FUNCTION_BLOCK XtsHardware
VAR_INPUT
END_VAR
VAR_OUTPUT
	XtsHardwareOK : BOOL;
	Xts48VStanding : BOOL;
	Xts24VStanding : BOOL;
END_VAR
VAR
	XtsIoEnvironment : Tc3_XTS_Utility.FB_TcIoXtsEnvironment;
	bInit: BOOL;
	bMoverIdDetectionError		: BOOL;
	bMoverIdDetectionActive		: BOOL;
	bMoverIdDetected : BOOL;
	f24V: ARRAY[1..nModuleNumber] OF LREAL;
	f48V: ARRAY[1..nModuleNumber] OF LREAL;
	CurrentLive : ARRAY[1..nModuleNumber] OF LREAL;
	MaxCurrent : ARRAY [1..nModuleNumber] OF DINT;
	nModuleCounter : INT := 1;
	nForCounter1 : UDINT;
	i: INT;
	State :(
        Init,                                               
		Redetect,
		MoversValid,                                 
        AllMoversFound,
		MoverIdDetection,
		XTSMode,
		CheckModuleVoltages,
		HWReady);
	Logger : TcMessage_Ext;
END_VAR
VAR CONSTANT
	nModuleNumber  : INT := 16;
END_VAR

IF NOT bInit THEN
	IF XtsIoEnvironment.Init(TRUE) THEN
		XtsIoEnvironment.Init(FALSE);
		bInit := TRUE;
	END_IF
	RETURN;
END_IF

CASE State OF
	Init:
		IF GetActiveTracks() THEN
			State := Redetect;
		END_IF
		
	Redetect:
		IF TriggerMoverDetection() THEN
			State := MoversValid;
		END_IF
		
	MoversValid:
		IF getAllMoversValid() THEN
			State := AllMoversFound;
		END_IF
	
	AllMoversFound:
		IF getMoversDetected() THEN
			State := MoverIdDetection;
		END_IF
		
	MoverIdDetection:
		IF TriggerMoverID() THEN
			State := XtsMode;
		END_IF
	
	XtsMode:
		IF IsInSim() THEN
			State := HWReady;
		ELSE
			State := CheckModuleVoltages;
		END_IF
		
	CheckModuleVoltages:
		Xts48VStanding := TRUE;
		Xts24VStanding := TRUE;
		FOR i := 1 TO nModuleNumber DO
			IF f48V[i] < 46000 THEN
				Xts48VStanding := FALSE;
			END_IF
			IF f24V[i] < 22000 THEN
				Xts24VStanding := FALSE;
			END_IF
		END_FOR
		IF Xts24VStanding AND Xts48VStanding THEN
			State := HWReady;
		END_IF
	
	HWReady:
		XtsHardwareOK := TRUE;
END_CASE

//Logger();
getModuleInfoData();

METHOD PUBLIC GetActiveTracks : BOOL
VAR_INPUT
END_VAR
FOR nForCounter1:=1 TO XtsIoEnvironment.XpuTcIo(1).GetTrackCount() DO
	XtsIoEnvironment.XpuTcIo(1).TrackTcIo(UDINT_TO_UINT(nForCounter1)).SetIsIncludedInDetection(FALSE);
END_FOR

FOR nForCounter1:=1 TO XtsIoEnvironment.XpuTcIo(1).GetTrackCount() DO
	XtsIoEnvironment.XpuTcIo(1).TrackTcIo(UDINT_TO_UINT(nForCounter1)).SetIsIncludedInDetection(TRUE);
	Logger.Send(TC_EVENTS.XtsHardwareEvents.ActiveTracksAddedForDetection, UDINT_TO_STRING(XtsIoEnvironment.XpuTcIo(1).GetTrackCount()));
	GetActiveTracks := TRUE;
END_FOR
END_METHOD

METHOD getAllMoversValid : BOOL
VAR_INPUT
END_VAR
 IF XtsIoEnvironment.XpuTcIo(1).GetAreAllPositionsValid() THEN
	 getAllMoversValid := TRUE;
	 Logger.Send(TC_EVENTS.XtsHardwareEvents.AllMoversValid,'');
 END_IF
END_METHOD

METHOD getModuleInfoData : BOOL
VAR_INPUT
END_VAR
IF XtsIoEnvironment.XpuTcIo(1).PartTcIo(1).ModuleCoE(nModuleCounter).InfoData.Update() THEN
	CurrentLive[nModuleCounter]:=XtsIoEnvironment.XpuTcIo(1).PartTcIo(1).ModuleCoE(nModuleCounter).InfoData.OverallCurrent;
	MaxCurrent[nModuleCounter]:=XtsIoEnvironment.XpuTcIo(1).PartTcIo(1).ModuleCoE(nModuleCounter).InfoData.MaxOverallCurrentLast500ms;
	f24V[nModuleCounter]:=XtsIoEnvironment.XpuTcIo(1).PartTcIo(1).ModuleCoE(nModuleCounter).InfoData.AuxiliaryVoltage24V;
	f48V[nModuleCounter]:=XtsIoEnvironment.XpuTcIo(1).PartTcIo(1).ModuleCoE(nModuleCounter).InfoData.DcLinkVoltage;
	//Increase Module count
	IF nModuleCounter = nModuleNumber THEN
		nModuleCounter:=1;
	ELSE
		nModuleCounter:=nModuleCounter+1;
	END_IF
END_IF
END_METHOD

METHOD getMoversDetected : BOOL
VAR_INPUT
END_VAR
IF XtsIoEnvironment.XpuTcIo(1).GetDetectedMoverCount() = XtsIoEnvironment.XpuTcIo(1).GetExpectedMoverCount() THEN
	getMoversDetected := TRUE;
	Logger.Send(TC_EVENTS.XtsHardwareEvents.ExpectedMoversDetected,UDINT_TO_STRING(XtsIoEnvironment.XpuTcIo(1).GetExpectedMoverCount()));
ELSE
	getMoversDetected := FALSE;
	Logger.Send(TC_EVENTS.XtsHardwareEvents.ExpectedMoversNotFound,'');
END_IF
END_METHOD

METHOD IsInSim : BOOL
VAR_INPUT
END_VAR
IF  XtsIoEnvironment.XpuTcIo(1).GetOperationMode() = OperationMode.Simulation THEN
	IsInSim := TRUE;
	Logger.Send(TC_EVENTS.XtsHardwareEvents.XtsInSimulationMode,'');
ELSE
	IsInSim := FALSE;
END_IF
END_METHOD

METHOD TriggerMoverDetection : BOOL
VAR_INPUT
END_VAR
XtsIoEnvironment.XpuTcIo(1).TriggerRedetection();
Logger.Send(TC_EVENTS.XtsHardwareEvents.MoverDetectionInitiated,'');
TriggerMoverDetection := true;
END_METHOD

METHOD TriggerMoverID : BOOL
VAR_INPUT
END_VAR
// Mover1 Functionality		
// Check if "MoverIdDetectionMode" has been activated under the XtsProcessingUnit object.
IF XtsIoEnvironment.XpuTcIo(1).GetMoverIdDetectionMode() = E_MoverIdDetectionMode.Mover1
	OR XtsIoEnvironment.XpuTcIo(1).GetMoverIdDetectionMode() = 2 THEN

	// Check if the "MoverIdDetection" has already been started or the Mover1 was found.
	IF NOT (bMoverIdDetectionActive OR bMoverIdDetected) THEN
		// Trigger the "MoverIdDetection".
		XtsIoEnvironment.XpuTcIo(1).TriggerMoverIdDetection();
		Logger.Send(TC_EVENTS.XtsHardwareEvents.Mover1DetectionStarted,'');
	END_IF

	// Check for error or success of "MoverIdDetection".
	bMoverIdDetectionError 	:= XtsIoEnvironment.XpuTcIo(1).GetHasMoverIdDetectionError();
	bMoverIdDetected 	:= XtsIoEnvironment.XpuTcIo(1).GetIsMoverIdDetectionValid();
	bMoverIdDetectionActive	:= XtsIoEnvironment.XpuTcIo(1).GetIsMoverIdDetectionActive();
	
	// If the detection has an error, check for errors in output and try again.
	IF bMoverIdDetectionError THEN
		Logger.Send(TC_EVENTS.XtsHardwareEvents.Mover1DetectionFailed,'');
		RETURN; 
	END_IF

	// Do not process any further until the "MoverId" was deteced.
	IF NOT bMoverIdDetected THEN
		RETURN;
	END_IF	
	TriggerMoverID := TRUE;	
	Logger.Send(TC_EVENTS.XtsHardwareEvents.Mover1DetectionComplete,'');
ELSE
	TriggerMoverID := TRUE;
	Logger.Send(TC_EVENTS.XtsHardwareEvents.StandardMoverNumberingComplete,'');
END_IF
END_METHOD

END_FUNCTION_BLOCK

(* stored: Version 1.1.0.1, ProductVersion 3.1.4024.11
   POU XtsHardware: Id {fdc8b717-d16e-40a4-b579-c07cec9aa7e9}, SpecialFunc None
   Method GetActiveTracks: Id {ef675147-48c6-4156-bca7-ee67e48b4aaa}
   Method getAllMoversValid: Id {ae944bc3-2c4d-4e0e-be98-33dfbe9c20d4}
   Method getModuleInfoData: Id {5df1d418-67cd-4681-b784-eb84b54fcac5}
   Method getMoversDetected: Id {812da94e-a8c0-4d51-9f58-8d59861ca284}
   Method IsInSim: Id {de7f62a4-75e4-488e-905d-35dc6644068b}
   Method TriggerMoverDetection: Id {31f9ff4a-273c-4d84-b7c3-87644d344482}
   Method TriggerMoverID: Id {fba9ec64-a56d-44cb-8f57-71a89622c1d8} *)
